FUNCTION_BLOCK FB_Co2FlowModelDeviationHandler
VAR_INPUT
	currentFlow : REAL;
	modeledFlow : REAL;
END_VAR
VAR_OUTPUT
	deviationPercentage : DINT;
END_VAR
VAR
	delta : REAL;
END_VAR


IF currentFlow <> 0 THEN
	delta := modeledFlow / currentFlow;
	
	IF delta < 0 THEN
		deviationPercentage := TO_DINT(delta*100);
	ELSE
		deviationPercentage := TO_DINT(-(100 - delta*100));
	END_IF
	
ELSE
	currentFlow := 0;
END_IF

END_FUNCTION_BLOCK

(* stored: Version 1.1.0.1, ProductVersion 3.1.4024.9
   POU FB_Co2FlowModelDeviationHandler: Id {f2cdafab-1b1c-4e4c-8880-93fc7a57225e}, SpecialFunc None *)
